// TIA Portal V20 export
FUNCTION_BLOCK "FB_Maintenances"   // FB473, SCL
{ S7_Optimized_Access := 'TRUE' }
// stored: AutoNumber false, MemoryReserve 100, SetENOAutomatically false
   VAR
      sCheckMachine : "FB_Maintenance";   // Message: Check Laser optical path (84h)
      sReplaceAirConditioningFilter { S7_SetPoint := 'True'} : "FB_Maintenance";   // Message: Clean the fairing (200 h)
      sMachineCooling_ReplaceWaterFilter { S7_SetPoint := 'True'} : "FB_Maintenance";   // Message: Clean the sheet metal (200 h)
      sTermotekChiller_ChangeFilterAndWater { S7_SetPoint := 'True'} : "FB_Maintenance";   // Message: Clean the screens (200 h)
      sCheckSafetySystem { S7_SetPoint := 'True'} : "FB_Maintenance";   // Message: Check the machine (200 h)
      sReplaceTipShellPeekGripper { S7_SetPoint := 'True'} : "FB_Maintenance";   // Message: Clean the clamping (200 h)
      sReplaceFiltersVacuumLoadingUnloading { S7_SetPoint := 'True'} : "FB_Maintenance";   // Message: Check the filter of the Laser power unit (2000 h)
      sReplaceFiltersVacuumGenerator { S7_SetPoint := 'True'} : "FB_Maintenance";   // Message: Check the safety systems (2000 h)
      sReplaceFilterAirDryer { S7_SetPoint := 'True'} : "FB_Maintenance";   // Message: Grease the X axis (1 y)
      sReplace5umFilter { S7_SetPoint := 'True'} : "FB_Maintenance";   // Message: Grease the Y axis (1 y)
      sReplace01umFilter { S7_SetPoint := 'True'} : "FB_Maintenance";   // Message: Check the water level of the TERMOTEK cooler (24 h)
      sReplaceActiveCarbonFilter { S7_SetPoint := 'True'} : "FB_Maintenance";   // Message: Clean the grid of the TERMOTEK cooler (24 h)
      sUTLExtraction_ReplaceParticleFilter { S7_SetPoint := 'True'} : "FB_Maintenance";   // Message: Check the operation of the condensate drain (24 h)
      sUTLExtraction_ReplaceFilterCassetteAndActiveCarbonFilter { S7_SetPoint := 'True'} : "FB_Maintenance";   // Message: Check the dew point under pressure (24 h)
      sReplaceSealOnSas { S7_SetPoint := 'True'} : "FB_Maintenance";   // Message: Clean the grid of the air dryer (24 h)
      sGreaseAxes { S7_SetPoint := 'True'} : "FB_Maintenance";   // Message: Replace the line filter of the air dryer (600 h)
      sMaintenance_16 { S7_SetPoint := 'True'} : "FB_Maintenance";   // Message: Replace 5 µm filter cartridge (600 h)
      sMaintenance_17 { S7_SetPoint := 'True'} : "FB_Maintenance";   // Message: Replace 0.01 µm filter cartridge (600 h)
      sMaintenance_18 { S7_SetPoint := 'True'} : "FB_Maintenance";   // Message: Replace the particles filter of the suction system (1000 h)
      sMaintenance_19 { S7_SetPoint := 'True'} : "FB_Maintenance";   // Message: Replace the filtration cassette AND the actived carbon of the suction system (1000 h)
      sMaintenance_20 { S7_SetPoint := 'True'} : "FB_Maintenance";   // Message: Replace the air conditioning filter (1000 h)
      sMaintenance_21 { S7_SetPoint := 'True'} : "FB_Maintenance";   // Message: Replace the TERMOTEK cooler filter (2000 h)
      sMaintenance_22 { S7_SetPoint := 'True'} : "FB_Maintenance";   // Message: Replace the water of the TERMOTEK cooler (2000 h)
      sMaintenance_23 { S7_SetPoint := 'True'} : "FB_Maintenance";   // Message: Spare
      sMaintenance_24 { S7_SetPoint := 'True'} : "FB_Maintenance";   // Message: Spare
      sMaintenance_25 { S7_SetPoint := 'True'} : "FB_Maintenance";   // Message: Spare
      sMaintenance_26 { S7_SetPoint := 'True'} : "FB_Maintenance";   // Message: Spare
      sMaintenance_27 { S7_SetPoint := 'True'} : "FB_Maintenance";   // Message: Spare
      sMaintenance_28 { S7_SetPoint := 'True'} : "FB_Maintenance";   // Message: Spare
      sMaintenance_29 { S7_SetPoint := 'True'} : "FB_Maintenance";   // Message: Spare
      sMaintenance_30 { S7_SetPoint := 'True'} : "FB_Maintenance";   // Message: Spare
      sMaintenance_31 { S7_SetPoint := 'True'} : "FB_Maintenance";   // Message: Spare
      sMaintenance_32 { S7_SetPoint := 'True'} : "FB_Maintenance";   // Message: Spare
      sMaintenance_33 { S7_SetPoint := 'True'} : "FB_Maintenance";   // Message: Spare
      sMaintenance_34 { S7_SetPoint := 'True'} : "FB_Maintenance";   // Message: Spare
      sMaintenance_35 { S7_SetPoint := 'True'} : "FB_Maintenance";   // Message: Spare
      sMaintenance_36 { S7_SetPoint := 'True'} : "FB_Maintenance";   // Message: Spare
      sMaintenance_37 { S7_SetPoint := 'True'} : "FB_Maintenance";   // Message: Spare
      sMaintenance_38 { S7_SetPoint := 'True'} : "FB_Maintenance";   // Message: Spare
      sMaintenance_39 { S7_SetPoint := 'True'} : "FB_Maintenance";   // Message: Spare
      sMaintenance_40 { S7_SetPoint := 'True'} : "FB_Maintenance";   // Message: Spare
      sMaintenance_41 { S7_SetPoint := 'True'} : "FB_Maintenance";   // Message: Spare
      sMaintenance_42 { S7_SetPoint := 'True'} : "FB_Maintenance";   // Message: Spare
      sMaintenance_43 { S7_SetPoint := 'True'} : "FB_Maintenance";   // Message: Spare
      sMaintenance_44 { S7_SetPoint := 'True'} : "FB_Maintenance";   // Message: Spare
      sMaintenance_45 { S7_SetPoint := 'True'} : "FB_Maintenance";   // Message: Spare
      sMaintenance_46 { S7_SetPoint := 'True'} : "FB_Maintenance";   // Message: Spare
      sMaintenance_47 { S7_SetPoint := 'True'} : "FB_Maintenance";   // Message: Spare
      sMaintenance_48 { S7_SetPoint := 'True'} : "FB_Maintenance";   // Message: Spare
      sMaintenance_49 { S7_SetPoint := 'True'} : "FB_Maintenance";   // Message: Spare
      sMaintenance_50 { S7_SetPoint := 'True'} : "FB_Maintenance";   // Message: Spare
      sMaintenance_51 { S7_SetPoint := 'True'} : "FB_Maintenance";   // Message: Spare
      sMaintenance_52 { S7_SetPoint := 'True'} : "FB_Maintenance";   // Message: Spare
      sMaintenance_53 { S7_SetPoint := 'True'} : "FB_Maintenance";   // Message: Spare
      sMaintenance_54 { S7_SetPoint := 'True'} : "FB_Maintenance";   // Message: Spare
      sMaintenance_55 { S7_SetPoint := 'True'} : "FB_Maintenance";   // Message: Spare
      sMaintenance_56 { S7_SetPoint := 'True'} : "FB_Maintenance";   // Message: Spare
      sMaintenance_57 { S7_SetPoint := 'True'} : "FB_Maintenance";   // Message: Spare
      sMaintenance_58 { S7_SetPoint := 'True'} : "FB_Maintenance";   // Message: Spare
      sMaintenance_59 { S7_SetPoint := 'True'} : "FB_Maintenance";   // Message: Spare
      sMaintenance_60 { S7_SetPoint := 'True'} : "FB_Maintenance";   // Message: Spare
      sMaintenance_61 { S7_SetPoint := 'True'} : "FB_Maintenance";   // Message: Spare
      sMaintenance_62 { S7_SetPoint := 'True'} : "FB_Maintenance";   // Message: Spare
      sMaintenance_63 { S7_SetPoint := 'True'} : "FB_Maintenance";   // Message: Spare
   END_VAR
BEGIN
   REGION Description header 
       //==================================================================================
       // POSALUX Swiss SA / (C) Copyright 2024
       //----------------------------------------------------------------------------------
       // Title: Maintenance
       // Comment/Function: Liste des apparaeils à controler dans la Liste des équipements 
       //                   pour la maintenance préventive  
       //
       // Author: Gowsigan SRITHARAN
       // Engineering: TIA Portal v17
       //----------------------------------------------------------------------------------
       // Change log table:
       // Version  | Date     | Expert in charge | Changes applied
       // ---------|----------|------------------|------------------------------------
       // 00.00.01 | 20250912 | WFA              | First released version
       // ==================================================================================
   END_REGION

   REGION 200 hours
           // Check the machine
           #sCheckMachine(iIncrementEnable := "LBP_Chan1".E_ProgRunning,
                          iID := 101,
                          ioOPC := "DB_OPC_Maintenance".Tasks[1],
                          ioAlarm := "LBP_AlarmMsgs".UserA[30].A70UUxx[00],
                          ioWarning := "LBP_AlarmMsgs".UserA[30].A70UUxx[32]);
      END_REGION

      REGION 1000 hours
           // Replace the air conditioning filter
           #sReplaceAirConditioningFilter(iIncrementEnable := "LBP_Chan1".E_ProgRunning,
                                          iID := 201,
                                          ioOPC := "DB_OPC_Maintenance".Tasks[2],
                                          ioAlarm := "LBP_AlarmMsgs".UserA[30].A70UUxx[01],
                                          ioWarning := "LBP_AlarmMsgs".UserA[30].A70UUxx[33]);

           // Machine cooling: replace water filter
           #sMachineCooling_ReplaceWaterFilter(iIncrementEnable := "LBP_Chan1".E_ProgRunning,
                                               iID := 202,
                                               ioOPC := "DB_OPC_Maintenance".Tasks[3],
                                               ioAlarm := "LBP_AlarmMsgs".UserA[30].A70UUxx[02],
                                               ioWarning := "LBP_AlarmMsgs".UserA[30].A70UUxx[34]);
      END_REGION

      REGION 2000 hours
          // Termotek chiller: change filter and water
          #sTermotekChiller_ChangeFilterAndWater(iIncrementEnable := "LBP_Chan1".E_ProgRunning,
                                                 iID := 301,
                                                 ioOPC := "DB_OPC_Maintenance".Tasks[4],
                                                 ioAlarm := "LBP_AlarmMsgs".UserA[30].A70UUxx[03],
                                                 ioWarning := "LBP_AlarmMsgs".UserA[30].A70UUxx[35]);

           // Check the safety system
           #sCheckSafetySystem(iIncrementEnable := "LBP_Chan1".E_ProgRunning,
                               iID := 302,
                               ioOPC := "DB_OPC_Maintenance".Tasks[5],
                               ioAlarm := "LBP_AlarmMsgs".UserA[30].A70UUxx[04],
                               ioWarning := "LBP_AlarmMsgs".UserA[30].A70UUxx[36]);

           // Replace the tip-shell PEEK gripper
           #sReplaceTipShellPeekGripper(iIncrementEnable := "LBP_Chan1".E_ProgRunning,
                                        iID := 303,
                                        ioOPC := "DB_OPC_Maintenance".Tasks[6],
                                        ioAlarm := "LBP_AlarmMsgs".UserA[30].A70UUxx[05],
                                        ioWarning := "LBP_AlarmMsgs".UserA[30].A70UUxx[37]);
      END_REGION

      REGION 3000 hours
           // Replace the filters for the vacuum of the loading/unloading
           #sReplaceFiltersVacuumLoadingUnloading(iIncrementEnable := "LBP_Chan1".E_ProgRunning,
                                                  iID := 401,
                                                  ioOPC := "DB_OPC_Maintenance".Tasks[7],
                                                  ioAlarm := "LBP_AlarmMsgs".UserA[30].A70UUxx[06],
                                                  ioWarning := "LBP_AlarmMsgs".UserA[30].A70UUxx[38]);

           // Replace the filters of the vacuum generator VADM
           #sReplaceFiltersVacuumGenerator(iIncrementEnable := "LBP_Chan1".E_ProgRunning,
                                           iID := 402,
                                           ioOPC := "DB_OPC_Maintenance".Tasks[8],
                                           ioAlarm := "LBP_AlarmMsgs".UserA[30].A70UUxx[07],
                                           ioWarning := "LBP_AlarmMsgs".UserA[30].A70UUxx[39]);
      END_REGION

      REGION 4000 hours
           // Replace the fine filter of the air dryer
           #sReplaceFilterAirDryer(iIncrementEnable := "LBP_Chan1".E_ProgRunning,
                                   iID := 501,
                                   ioOPC := "DB_OPC_Maintenance".Tasks[9],
                                   ioAlarm := "LBP_AlarmMsgs".UserA[30].A70UUxx[08],
                                   ioWarning := "LBP_AlarmMsgs".UserA[30].A70UUxx[40]);

           // Replace the 5 μm filter
           #sReplace5umFilter(iIncrementEnable := "LBP_Chan1".E_ProgRunning,
                              iID := 502,
                              ioOPC := "DB_OPC_Maintenance".Tasks[10],
                              ioAlarm := "LBP_AlarmMsgs".UserA[30].A70UUxx[09],
                              ioWarning := "LBP_AlarmMsgs".UserA[30].A70UUxx[41]);

          // Replace the 0.1 μm filter
         #sReplace01umFilter(iIncrementEnable := "LBP_Chan1".E_ProgRunning,
                             iID := 503,
                             ioOPC := "DB_OPC_Maintenance".Tasks[11],
                             ioAlarm := "LBP_AlarmMsgs".UserA[30].A70UUxx[10],
                             ioWarning := "LBP_AlarmMsgs".UserA[30].A70UUxx[42]);

           // Replace the active carbon filter
           #sReplaceActiveCarbonFilter(iIncrementEnable := "LBP_Chan1".E_ProgRunning,
                                       iID := 504,
                                       ioOPC := "DB_OPC_Maintenance".Tasks[12],
                                       ioAlarm := "LBP_AlarmMsgs".UserA[30].A70UUxx[11],
                                       ioWarning := "LBP_AlarmMsgs".UserA[30].A70UUxx[43]);

           // UTL extraction: replace particle filter
           #sUTLExtraction_ReplaceParticleFilter(iIncrementEnable := "LBP_Chan1".E_ProgRunning,
                                                 iID := 505,
                                                 ioOPC := "DB_OPC_Maintenance".Tasks[13],
                                                 ioAlarm := "LBP_AlarmMsgs".UserA[30].A70UUxx[12],
                                                 ioWarning := "LBP_AlarmMsgs".UserA[30].A70UUxx[44]);

           // UTL extraction: replace filter cassette and active carbon filter
           #sUTLExtraction_ReplaceFilterCassetteAndActiveCarbonFilter(iIncrementEnable := "LBP_Chan1".E_ProgRunning,
                                                                      iID := 506,
                                                                      ioOPC := "DB_OPC_Maintenance".Tasks[14],
                                                                      ioAlarm := "LBP_AlarmMsgs".UserA[30].A70UUxx[13],
                                                                      ioWarning := "LBP_AlarmMsgs".UserA[30].A70UUxx[45]);

      END_REGION

      REGION 6000 hours
           // Replace the seal on the air lock door (SAS)
           #sReplaceSealOnSas(iIncrementEnable := "LBP_Chan1".E_ProgRunning,
                              iID := 601,
                              ioOPC := "DB_OPC_Maintenance".Tasks[15],
                              ioAlarm := "LBP_AlarmMsgs".UserA[30].A70UUxx[14],
                              ioWarning := "LBP_AlarmMsgs".UserA[30].A70UUxx[46]);

           // Grease the axes
           #sGreaseAxes(iIncrementEnable := "LBP_Chan1".E_ProgRunning,
                        iID := 602,
                        ioOPC := "DB_OPC_Maintenance".Tasks[16],
                        ioAlarm := "LBP_AlarmMsgs".UserA[30].A70UUxx[15],
                        ioWarning := "LBP_AlarmMsgs".UserA[30].A70UUxx[47]);
      END_REGION
END_FUNCTION_BLOCK
